// TIA Portal project "Marcha_Parada_S_R" (V13)

(* hardware
DEVICE "S7-1200 station_1"  S7-1200 Station
   slot 0: "Rack_0"  Rack  V1.0
   slot 1: "PLC_1"  CPU 1214C AC/DC/Rly  6ES7 214-1BE30-0XB0  V2.2
*)

// ===== PLC "PLC_1"  CPU 1214C AC/DC/Rly =====

VAR_GLOBAL   // PLC tag table "Tabla de variables estándar"
   "MARCHA" AT %I0.1 : Bool;
   "PARO" AT %I0.2 : Bool;
   "MOTOR" AT %Q0.0 : Bool;
   "T_MARCHA" AT %Q0.1 : Bool;
   "T_PARO" AT %Q0.2 : Bool;
   "M_P" AT %M10.1 : Bool;
   "M_N" AT %M10.2 : Bool;
END_VAR

ORGANIZATION_BLOCK "Main"   // OB1, LAD, ProgramCycle
TITLE = "Main Program Sweep (Cycle)"
{ S7_Optimized_Access := 'FALSE' }
VERSION : 0.1
   VAR_TEMP   // added for the SCL form of the ladder/FBD networks
      _w1 : Bool;
      _w2 : Bool;
   END_VAR
BEGIN

REGION Network 1
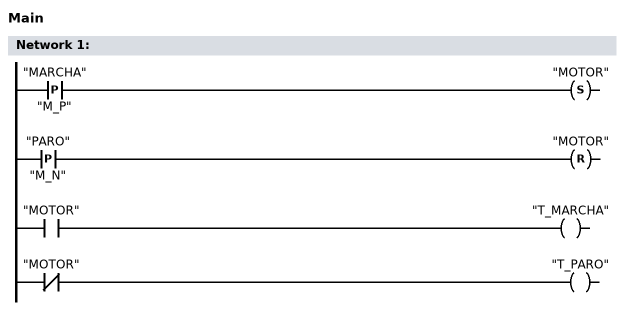
   RUNG wire#powerrail
      P_Contact(operand := "MARCHA", bit := "M_P")
      S_Coil( "MOTOR" )
   END_RUNG
   RUNG wire#powerrail
      P_Contact(operand := "PARO", bit := "M_N")
      R_Coil( "MOTOR" )
   END_RUNG
   RUNG wire#powerrail
      Contact( "MOTOR" )
      Coil( "T_MARCHA" )
   END_RUNG
   RUNG wire#powerrail
      I_Contact( "MOTOR" )
      Coil( "T_PARO" )
   END_RUNG
   // the same network as SCL:
   #_w1 := "MARCHA" AND NOT "M_P";   // rising edge of "MARCHA"
   "M_P" := "MARCHA";
   IF #_w1 THEN "MOTOR" := TRUE; END_IF;
   #_w2 := "PARO" AND NOT "M_N";   // rising edge of "PARO"
   "M_N" := "PARO";
   IF #_w2 THEN "MOTOR" := FALSE; END_IF;
   "T_MARCHA" := "MOTOR";
   "T_PARO" := NOT "MOTOR";
END_REGION
END_ORGANIZATION_BLOCK